# EPICS IOC start-up script: iocsh/ethercatmcEL6688-EL1252-PTP.iocsh
ethercatmcCreateAsynParam $(MOTOR_PORT) TS_NS             Int32

dbLoadRecords("ethercatmcEL6688-EL1252-PTP.template", "SYSPFX=$(SYSPFX), REG_NAME=$(REG_NAME), MOTOR_PORT=$(MOTOR_PORT)")
